// Something that carries a human-readable name.
//
// Extracted because a suite needs a label in two unrelated roles - as the thing
// the sequencer drives, and as the thing an observer reads counts from - and
// declaring it twice would let the two drift apart.
INTERFACE I_Labelled EXTENDS __SYSTEM.IQueryInterface

// The name that appears in results. Stable across renames of the underlying
// instance, because it is supplied rather than derived.
PROPERTY Label : T_MaxString
GET
END_GET
END_PROPERTY

END_INTERFACE

(* stored: Version 1.1.0.1
   Itf I_Labelled: Id {6f7abda0-ad0a-422a-ad6f-6e8fb2c93470}
   Property Label: Id {2820da08-fae7-45ea-a9e0-97a41685d5c7}
   Get Get: Id {2ad70b13-51b4-4e1c-aa61-adac70acd6ba} *)
